// TIA Portal project "Carrello_CTUD" (V15.1)

(* hardware
DEVICE "S7-1200 station_1"  S7-1200 Station
   slot 0: "Telaio di montaggio_0"  S7-1200 Rack  Rack  V1.0
   slot 1: "PLC_1"  CPU 1214C DC/DC/DC  6ES7 214-1AG40-0XB0  V4.2
*)

// ===== PLC "PLC_1"  CPU 1214C DC/DC/DC =====

VAR_GLOBAL   // PLC tag table "Tabella delle variabili standard"
   "SI" AT %I0.0 : Bool;
   "SQ" AT %I0.1 : Bool;
   "motore" AT %Q0.0 : Bool;
   "contatore" AT %MW0 : Int;
   "reset" AT %I0.2 : Bool;
   "preset" AT %I0.3 : Bool;
END_VAR

VAR_GLOBAL CONSTANT   // PLC tag table "Tabella delle variabili standard"
   "valoreIniziale" : Int := 10;
   "valoreZero" : Int := 0;
END_VAR

// folder: System blocks/Program resources

DATA_BLOCK "IEC_Counter_0_DB"   // DB1
{ S7_Optimized_Access := 'TRUE' }
AUTHOR : Simatic
FAMILY : IEC
NAME : CNTR
VERSION : 1.0
// stored: InstanceOfName IEC_COUNTER
"IEC_COUNTER"
BEGIN
END_DATA_BLOCK

// folder: (top level)

ORGANIZATION_BLOCK "Main"   // OB1, LAD, ProgramCycle
TITLE = "Main Program Sweep (Cycle)"
{ S7_Optimized_Access := 'TRUE' }
VERSION : 0.1
   VAR_INPUT
      Initial_Call : Bool;   // Initial call of this OB
      Remanence : Bool;   // =True, if remanent data are available
   END_VAR
BEGIN

REGION Network 1
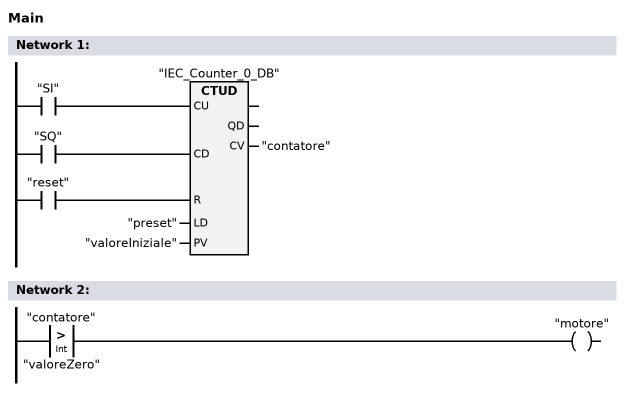
   "IEC_Counter_0_DB".CTUD(CU := "SI",
                           CD := "SQ",
                           R := "reset",
                           LD := "preset",
                           PV := "valoreIniziale",
                           CV => "contatore");
END_REGION

REGION Network 2
   RUNG wire#powerrail
      { S7_Templates := "SrcType := Int" } GT_Contact(in1 := "contatore", in2 := "valoreZero")
      Coil( "motore" )
   END_RUNG
   // the same network as SCL:
   "motore" := "contatore" > "valoreZero";
END_REGION
END_ORGANIZATION_BLOCK